FUNCTION_BLOCK AlgorithmWithTemporaryVariables
  (* Standard: 61499-2 *)
  (* Version 0.0, 4/15/2022, Radimir.Sorokin, FBME, Test *)
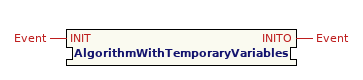
  EVENT_INPUT
    INIT;
  END_EVENT
  EVENT_OUTPUT
    INITO;
  END_EVENT
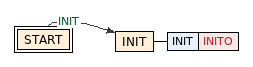
  EC_STATES
    START;
    INIT : INIT -> INITO;
  END_STATES
  EC_TRANSITIONS
    START TO INIT := INIT;
  END_TRANSITIONS
  ALGORITHM INIT IN ST:
VAR
	temp : INT;
END_VAR
tempt := 0;
temp := temp + 1;
  END_ALGORITHM
END_FUNCTION_BLOCK
